FUNCTION_BLOCK SLOT_SET_TRAJ_OFFSET (* Sets trajectory offset distances from centerline *)
  (* Standard: 61499-2 *)
  (* Version 1.0, 27-05-12, GASR, Universidade do Estado de Santa Catarina *)
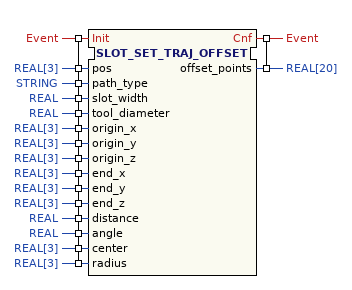
  EVENT_INPUT
    Init WITH pos, path_type, slot_width, tool_diameter, origin_x, origin_y, origin_z, end_x, end_y, end_z, distance, angle, center, radius;
  END_EVENT
  EVENT_OUTPUT
    Cnf WITH offset_points;
  END_EVENT
  VAR_INPUT
    pos : ARRAY [0..2] OF REAL;
    path_type : STRING;
    slot_width : REAL;
    tool_diameter : REAL;
    origin_x : ARRAY [0..2] OF REAL;
    origin_y : ARRAY [0..2] OF REAL;
    origin_z : ARRAY [0..2] OF REAL;
    end_x : ARRAY [0..2] OF REAL;
    end_y : ARRAY [0..2] OF REAL;
    end_z : ARRAY [0..2] OF REAL;
    distance : REAL;
    angle : REAL;
    center : ARRAY [0..2] OF REAL;
    radius : ARRAY [0..2] OF REAL;
  END_VAR
  VAR_OUTPUT
    offset_points : ARRAY [0..19] OF REAL; (* offset points list *)
  END_VAR
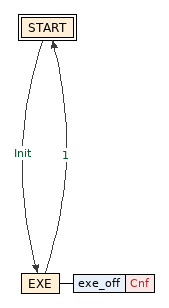
  EC_STATES
    START;
    EXE : exe_off -> Cnf;
  END_STATES
  EC_TRANSITIONS
    START TO EXE := Init;
    EXE TO START := 1;
  END_TRANSITIONS
  ALGORITHM exe_off IN Lua:
local offset = (slot_width/tool_diameter)
print( 'po', path_type, offset, slot_width, tool_diameter, 'center', center[1], center[2], center[3], 'pos', pos[1], pos[2], pos[3] )
print( 'VECTORS', 'o_y', origin_y[1], origin_y[2], origin_y[3] )
if not( offset > 1 ) then
    if( path_type == 'LINEAR_PATH' ) then
        offset_points[1] = { pos[1], pos[2], pos[3] }
        offset_points[2] = { pos[1] + origin_x[1]*distance, pos[2] + origin_x[2]*distance, pos[3] + origin_x[3]*distance }
    elseif( path_type == 'COMPLETE_CIRCULAR_PATH' ) then
        offset_points[1] = { pos[1], pos[2], pos[3] }
        offset_points[2] = { center[1], center[2], center[3], 360, radius, origin_z[1], origin_z[2], origin_z[3] }
    elseif( path_type == 'PARTIAL_CIRCULAR_PATH' ) then
        offset_points[1] = { pos[1], pos[2], pos[3] }
        offset_points[2] = { center[1], center[2], center[3], angle, radius, origin_z[1], origin_z[2], origin_z[3] }
        offset_points[3] = { center[1], center[2], center[3], -angle, radius, origin_z[1], origin_z[2], origin_z[3] }
    end
else
    local off_p = {}
    local off_int = math.floor( offset )
	local off_float = offset - off_int
	for i = 1, off_int do
        off_p[i] = 1
    end
    if( off_float > 0 ) then
        off_p[ #off_p + 1 ] = off_float
    end
    offset_points[1] = { (pos[1] - origin_y[1]*((slot_width/2 - (tool_diameter/2)))), (pos[2] - origin_y[2]*((slot_width/2 - (tool_diameter/2)))), (pos[3] - origin_y[3]*((slot_width/2 - (tool_diameter/2)))) }
    local status = 'going'
    for i = 1, (#off_p - 1) do
        if( path_type == 'LINEAR_PATH' ) then
            if( status == 'going' ) then
                offset_points[ 2*i ] = { offset_points[ 2*i - 1 ][1] + origin_x[1]*distance, offset_points[ 2*i - 1 ][2] + origin_x[2]*distance, offset_points[ 2*i - 1 ][3] + origin_x[3]*distance }
                status = 'coming'
            else
                offset_points[ 2*i ] = { offset_points[ 2*i - 1 ][1] - origin_x[1]*distance, offset_points[ 2*i - 1 ][2] - origin_x[2]*distance, offset_points[ 2*i - 1 ][3] - origin_x[3]*distance }
                status = 'going'
            end
        offset_points[ 2*i + 1 ] = { offset_points[ 2*i ][1] + origin_y[1]*(tool_diameter)*off_p[i], offset_points[ 2*i ][2] + origin_y[2]*(tool_diameter)*off_p[i], offset_points[ 2*i ][3] + origin_y[3]*(tool_diameter)*off_p[i] }
	elseif( path_type == 'COMPLETE_CIRCULAR_PATH' ) then
            local prov_radius = ( (offset_points[ 2*i - 1 ][1] - center[1])^2 + (offset_points[ 2*i - 1 ][2] - center[2])^2 + (offset_points[ 2*i - 1 ][3] - center[3])^2 )^0.5
            print( prov_radius, offset_points[ 2*i - 1 ][1], offset_points[ 2*i - 1 ][2], offset_points[ 2*i - 1 ][3], center[1], center[2], center[3] )
            if( status == 'going' ) then
                offset_points[ 2*i ] = { center[1], center[2], center[3], 360, prov_radius, origin_z[1], origin_z[2], origin_z[3] }
                print( #offset_points[ 2*i ] )
                status = 'coming'
            else
                offset_points[ 2*i ] = { center[1], center[2], center[3], -360, prov_radius, origin_z[1], origin_z[2], origin_z[3] }
                status = 'going'
            end
            print( 'VECTORS', 'o_y', off_p[i], offset_points[ 2*i ][1] + origin_y[1]*(tool_diameter)*off_p[i], origin_y[2], origin_y[3] )
            offset_points[ 2*i + 1 ] = { offset_points[ 2*i - 1][1] + origin_y[1]*(tool_diameter)*off_p[i + 1], offset_points[ 2*i - 1 ][2] + origin_y[2]*(tool_diameter)*off_p[i + 1], offset_points[ 2*i - 1 ][3] + origin_y[3]*(tool_diameter)*off_p[i + 1] }
        elseif( path_type == 'PARTIAL_CIRCULAR_PATH' ) then
            local prov_radius = ( (offset_points[ 3*i - 2 ][1] - center[1])^2 + (offset_points[ 3*i - 2 ][2] - center[2])^2 + (offset_points[ 3*i - 2 ][3] - center[3])^2 )^0.5
            print( 'prov_radius', prov_radius, offset_points[ 3*i - 2 ][1], offset_points[ 3*i - 2 ][2], offset_points[ 3*i - 2 ][3], center[1], center[2], center[3] )
            offset_points[ 3*i - 1 ] = { center[1], center[2], center[3], angle, prov_radius, origin_z[1], origin_z[2], origin_z[3] }
            offset_points[ 3*i ] = { center[1], center[2], center[3], -angle, prov_radius, origin_z[1], origin_z[2], origin_z[3] }
            offset_points[ 3*i + 1 ] = { (offset_points[ 3*i - 2 ][1] + origin_y[1]*(tool_diameter)*off_p[i + 1]),
                                 (offset_points[ 3*i - 2 ][2] + origin_y[2]*(tool_diameter)*off_p[i + 1]),
                                 (offset_points[ 3*i - 2 ][3] + origin_y[3]*(tool_diameter)*off_p[i + 1]) }
        end
    end
    if( path_type == 'LINEAR_PATH' ) then
        if( status == 'going' ) then
            offset_points[ 2*(#off_p) ] = { offset_points[ 2*(#off_p) - 1 ][1] + origin_x[1]*distance, offset_points[ 2*(#off_p) - 1 ][2] + origin_x[2]*distance, offset_points[ 2*(#off_p) - 1 ][3] + origin_x[3]*distance }
        else
            offset_points[ 2*(#off_p) ] = { offset_points[ 2*(#off_p) - 1 ][1] - origin_x[1]*distance, offset_points[ 2*(#off_p) - 1 ][2] - origin_x[2]*distance, offset_points[ 2*(#off_p) - 1 ][3] - origin_x[3]*distance }
        end
    elseif( path_type == 'COMPLETE_CIRCULAR_PATH' ) then
        local prov_radius = (( (offset_points[ 2*(#off_p) - 1 ][1] - center[1])^2 + (offset_points[ 2*(#off_p) - 1 ][2] - center[2])^2 + (offset_points[ 2*(#off_p) - 1 ][3] - center[3])^2 )^0.5)
        print( 'prov_radius', prov_radius  )
        if( status == 'going' ) then
            offset_points[ 2*(#off_p) ] = { center[1], center[2], center[3], 360, prov_radius, origin_z[1], origin_z[2], origin_z[3] }
        else
            offset_points[ 2*(#off_p) ] = { center[1], center[2], center[3], -360, prov_radius, origin_z[1], origin_z[2], origin_z[3] }
        end
    elseif( path_type == 'PARTIAL_CIRCULAR_PATH' ) then
        local prov_radius = (( (offset_points[ 3*(#off_p) - 2 ][1] - center[1])^2 + (offset_points[ 3*(#off_p) - 2 ][2] - center[2])^2 + (offset_points[ 3*(#off_p) - 2 ][3] - center[3])^2 )^0.5)
        offset_points[ 3*(#off_p) - 1 ] = { center[1], center[2], center[3], angle, prov_radius, origin_z[1], origin_z[2], origin_z[3] }
            offset_points[ 3*(#off_p) ] = { center[1], center[2], center[3], -angle, prov_radius, origin_z[1], origin_z[2], origin_z[3] }
    end
end
  END_ALGORITHM
END_FUNCTION_BLOCK
